// TIA Portal V16 export
// export: Created 2023-09-11T12:14:56.3982487Z, ExportSetting WithDefaults, DisplayName Totally Integrated Automation Portal, DisplayVersion V16 Update 6, DisplayName TIA Portal Version Control Interface, DisplayVersion V16 Update 2, DisplayName TIA Portal Openness, DisplayVersion V16 Update 6, DisplayName STEP 7 Professional, DisplayVersion V16 Update 6, DisplayName STEP 7 Safety, DisplayVersion V16, DisplayName WinCC Advanced, DisplayVersion V16 Update 6
DATA_BLOCK "Data_Czas_synch"   // DB32
{ S7_Optimized_Access := 'FALSE' }
VERSION : 0.1
// stored: AutoNumber false, DBAccessibleFromOPCUA true, IsOnlyStoredInLoadMemory false, IsWriteProtectedInAS false
   VAR
      Time_Local_read : DTL;
      Time_System_read : DTL;
      Time_System_write : DTL;
      zegar : Time_Of_Day;
      actTime : Real;
   END_VAR
BEGIN
END_DATA_BLOCK
